// TIA Portal V16 export
// export: Created 2024-12-03T15:41:46.0909211Z, ExportSetting WithReadOnly, DisplayName Totally Integrated Automation Portal, DisplayVersion V16 Update 6, DisplayName TIA Portal Version Control Interface, DisplayVersion V16 Update 2, DisplayName TIA Portal Openness, DisplayVersion V16 Update 6, DisplayName TIA Portal Teamcenter Gateway, DisplayVersion V16, DisplayName SINAMICS Startdrive Advanced, DisplayVersion V16 Update 5, DisplayName SINAMICS Startdrive G130, G150, S120, S150, SINAMICS MV, S210, DisplayVersion V16 Update 5, DisplayName SINAMICS Startdrive G110M, G120, G120C, G120D, G120P, G115D, DisplayVersion V16 Update 5, DisplayName STEP 7 Professional, DisplayVersion V16 Update 6, DisplayName STEP 7 Safety, DisplayVersion V16, DisplayName WinCC Advanced / Unified PC, DisplayVersion V16 Update 6
TYPE "VirtualEncoder_UDT"
// stored: CreationDate 2021-07-13T07:41:36.2278727Z, InterfaceModifiedDate 2021-04-04T08:21:35.5151954Z, IsConsistent true, LibraryConformanceStatus The object is library-conformant., ModifiedDate 2021-07-03T12:49:45.8681804Z
   STRUCT
      Distance_mm : Real;
      Speed_mm_ms : Real;
      Settings : Struct   // When the conveyor is running on baserelative it moves x M/min
         Base_M_min { S7_SetPoint := 'True'} : Real := 50.0;   // M/min base
         BaseRelative { S7_SetPoint := 'True'} : Real := 100.0;   // base relative %
      END_STRUCT;
   END_STRUCT;
END_TYPE
